FUNCTION F_astroRad2Dms : LREAL
VAR_INPUT
	dd:	LREAL;	// angle in radians
END_VAR
VAR
	value:		LREAL;
	degrees:	INT;
	minutes:	INT;
	seconds:	LREAL;
	
	sign:	int := 1;
END_VAR

IF dd < 0.0 THEN
	sign	:= -1;
	dd		:= -dd;
END_IF

value := dd / GCL.C_2PI * 360.0; 	// rad to degrees


degrees	:= TRUNC_INT(value);
minutes := TRUNC_INT((value - degrees)*60.0);
seconds := (value - degrees - minutes/60.0)*3600.0;

					
F_astroRad2Dms	:= (degrees * 10000 + minutes * 100 + seconds) * sign;

END_FUNCTION

(* stored: Version 1.1.0.1, ProductVersion 3.1.4024.10
   POU F_astroRad2Dms: Id {7c76b9a5-f6a3-40f7-8bab-0a23cf28a620}, SpecialFunc None *)
